KUKA KRL program: CVExample.src, CVExample.dat

--- CVExample.src ---
&ACCESS RVO
&REL 1
&PARAM EDITMASK = *
&PARAM TEMPLATE = C:\KRC\Roboter\Template\ExpertVorgabe
DEF CVExample( )

END

--- CVExample.dat ---
&ACCESS RVO
&REL 1
&PARAM EDITMASK = *
&PARAM TEMPLATE = C:\KRC\Roboter\Template\ExpertVorgabe
DEFDAT CVExample PUBLIC

int myvar = 123456879

ENDDAT
